// TIA Portal project "8m2" (V16)

(* hardware
DEVICE "S7-1200 station_1"  S7-1200 Station
   slot 0: "Rack_0"  S7-1200 Rack  Rack  V1.0
   slot 1: "PLC_1"  CPU 1212C AC/DC/Rly  6ES7 212-1BE40-0XB0  V4.4
*)

// ===== PLC "PLC_1"  CPU 1212C AC/DC/Rly =====

VAR_GLOBAL   // PLC tag table "Default tag table"
   "START" AT %I0.1 : Bool;
   "STOP" AT %I0.2 : Bool;
   "MOTOR1" AT %Q0.0 : Bool;
   "MOTOR2" AT %Q0.1 : Bool;
   "MOTOR3" AT %Q0.2 : Bool;
   "MARKER1" AT %M0.0 : Bool;
   "MARKER2" AT %M0.1 : Bool;
   "MARKER3" AT %M0.2 : Bool;
   "MARKER" AT %M0.3 : Bool;
   "X" AT %M0.4 : Bool;
END_VAR

// folder: System blocks/Program resources

DATA_BLOCK "TIMER1"   // DB1
{ S7_Optimized_Access := 'TRUE' }
AUTHOR : Simatic
FAMILY : IEC
NAME : IEC_TMR
VERSION : 1.0
// stored: InstanceOfName IEC_TIMER
"IEC_TIMER"
BEGIN
END_DATA_BLOCK

DATA_BLOCK "TIMER2"   // DB2
{ S7_Optimized_Access := 'TRUE' }
AUTHOR : Simatic
FAMILY : IEC
NAME : IEC_TMR
VERSION : 1.0
// stored: InstanceOfName IEC_TIMER
"IEC_TIMER"
BEGIN
END_DATA_BLOCK

DATA_BLOCK "TIMER3"   // DB3
{ S7_Optimized_Access := 'TRUE' }
AUTHOR : Simatic
FAMILY : IEC
NAME : IEC_TMR
VERSION : 1.0
// stored: InstanceOfName IEC_TIMER
"IEC_TIMER"
BEGIN
END_DATA_BLOCK

// folder: (top level)

ORGANIZATION_BLOCK "Main"   // OB1, LAD, ProgramCycle
TITLE = "Main Program Sweep (Cycle)"
{ S7_Optimized_Access := 'TRUE' }
VERSION : 0.1
   VAR_INPUT
      Initial_Call : Bool;   // Initial call of this OB
      Remanence : Bool;   // =True, if remanent data are available
   END_VAR
BEGIN

REGION Network 1
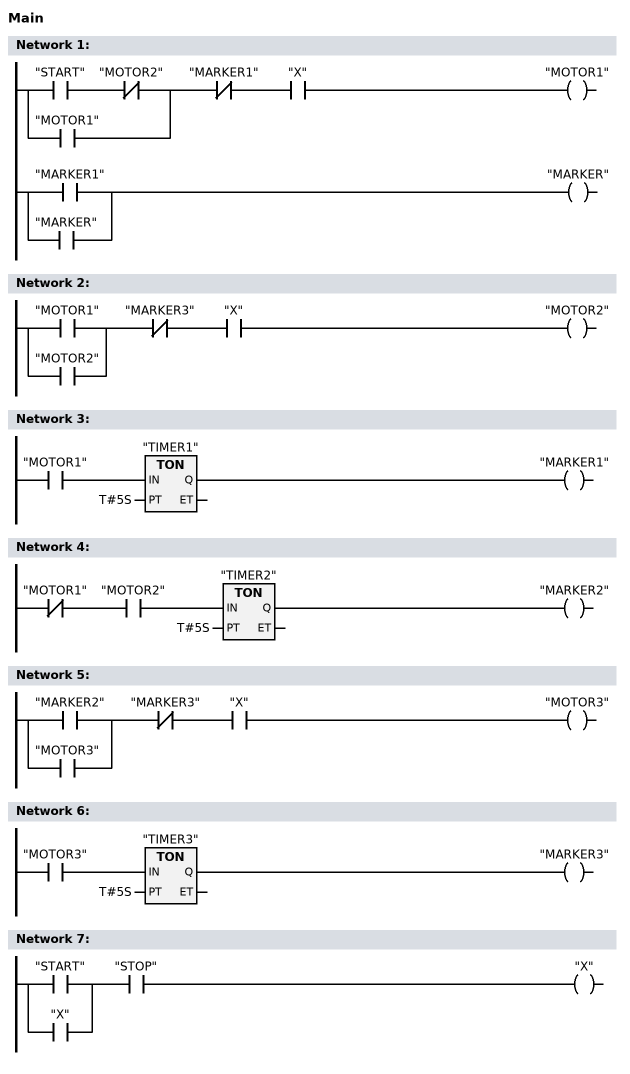
   RUNG wire#powerrail
      Contact( "START" )
      I_Contact( "MOTOR2" )
      wire#w1
      I_Contact( "MARKER1" )
      Contact( "X" )
      Coil( "MOTOR1" )
   END_RUNG
   RUNG wire#powerrail
      Contact( "MOTOR1" )
   END_RUNG wire#w1
   RUNG wire#powerrail
      Contact( "MARKER1" )
      wire#w2
      Coil( "MARKER" )
   END_RUNG
   RUNG wire#powerrail
      Contact( "MARKER" )
   END_RUNG wire#w2
   // the same network as SCL:
   "MOTOR1" := (("START" AND NOT "MOTOR2") OR "MOTOR1") AND NOT "MARKER1" AND "X";
   "MARKER" := "MARKER1" OR "MARKER";
END_REGION

REGION Network 2
   RUNG wire#powerrail
      Contact( "MOTOR1" )
      wire#w1
      I_Contact( "MARKER3" )
      Contact( "X" )
      Coil( "MOTOR2" )
   END_RUNG
   RUNG wire#powerrail
      Contact( "MOTOR2" )
   END_RUNG wire#w1
   // the same network as SCL:
   "MOTOR2" := ("MOTOR1" OR "MOTOR2") AND NOT "MARKER3" AND "X";
END_REGION

REGION Network 3
   "TIMER1".TON(IN := "MOTOR1", PT := T#5S);
   "MARKER1" := "TIMER1".Q;
END_REGION

REGION Network 4
   "TIMER2".TON(IN := NOT "MOTOR1" AND "MOTOR2", PT := T#5S);
   "MARKER2" := "TIMER2".Q;
END_REGION

REGION Network 5
   RUNG wire#powerrail
      Contact( "MARKER2" )
      wire#w1
      I_Contact( "MARKER3" )
      Contact( "X" )
      Coil( "MOTOR3" )
   END_RUNG
   RUNG wire#powerrail
      Contact( "MOTOR3" )
   END_RUNG wire#w1
   // the same network as SCL:
   "MOTOR3" := ("MARKER2" OR "MOTOR3") AND NOT "MARKER3" AND "X";
END_REGION

REGION Network 6
   "TIMER3".TON(IN := "MOTOR3", PT := T#5S);
   "MARKER3" := "TIMER3".Q;
END_REGION

REGION Network 7
   RUNG wire#powerrail
      Contact( "START" )
      wire#w1
      Contact( "STOP" )
      Coil( "X" )
   END_RUNG
   RUNG wire#powerrail
      Contact( "X" )
   END_RUNG wire#w1
   // the same network as SCL:
   "X" := ("START" OR "X") AND "STOP";
END_REGION
END_ORGANIZATION_BLOCK